TYPE ST_System :
STRUCT
	Inputs					: ST_System_In;			// System inputs
	Outputs					: ST_System_Out;		// System outputs
	SystemTime				: ST_TimeManagement;	// System time and pulses	
	PackMLState				: ST_PMLState;			// System PackML data
END_STRUCT
END_TYPE

(* stored: Version 1.1.0.1, ProductVersion 3.1.4024.3
   DUT ST_System: Id {e1e5d9de-91de-415b-9c43-7292cc00a990} *)
